FUNCTION_BLOCK ReadBsDeviationMax
VAR_INPUT
	nIdxGrp: UDINT;
	bStart: BOOL;
	pDest: POINTER TO UDINT;
END_VAR
VAR_OUTPUT
	Busy: BOOL;
	bErr: BOOL;
END_VAR
VAR
	fbRead: ADSREAD;
	bStarted: BOOL;
END_VAR

IF bStarted = FALSE THEN
   IF bStart = TRUE THEN
      bStarted := TRUE;
      bErr := FALSE;
      Busy := TRUE;
   END_IF
END_IF

IF bStarted THEN
   (* raising edge of Timer triggers read request *)
   fbRead( NetID := '', Port := 553, IdxGrp := nIdxGrp, IdxOffs := 16#00000064,
         LEN := 4, DestAddr := pDest, READ := bStarted, TMOUT := T#1s);
   IF NOT fbRead.Busy THEN
      (* There was an error in the execution of the read request *)
      IF fbRead.Err THEN
         bErr := TRUE;
      END_IF
      fbRead(READ := FALSE);    (* reset because of edge detection in FB ADSREAD *)
      bStarted := FALSE;
      Busy := FALSE;
   END_IF
END_IF

END_FUNCTION_BLOCK

(* stored: Version 1.1.0.1, ProductVersion 3.1.0.12
   POU ReadBsDeviationMax: Id {829f9ccc-a0fd-4048-9f1f-4390e9af290c} *)
